TYPE
	NW_BUF_LONG  : ARRAY[0..NETWORK_BUFFER_LONG_SIZE] OF BYTE;
END_TYPE

(* stored: Version 1.1.0.1, ProductVersion 3.1.4024.9
   DUT NW_BUF_LONG: Id {dbd5f6a9-6749-42a7-bdf2-4ee344480bfc} *)
